// TIA Portal V20 export
TYPE "LConSMC_typeTaper"
// Ein-/Ausgänge der Zugreduktion / In-/Outputs of the tension taper
// stored: Access Published
   STRUCT
      in { S7_SetPoint := 'True'} : "LConSMC_typeTaperInput";   // Eingänge des Bausteins Taper / Inputs for FB Taper
      out { S7_SetPoint := 'True'} : "LConSMC_typeTaperOutput";   // Ausgänge des Bausteins Taper / Outputs for FB Taper
   END_STRUCT;
END_TYPE
